// TIA Portal V19 export
DATA_BLOCK "ProcessAndPbAlarms"   // DB2
{ S7_Optimized_Access := 'TRUE' }
AUTHOR : FLA
FAMILY : UHT
VERSION : 1.0
// stored: AutoNumber false, MemoryReserve 0
   VAR
      "A" : Array[1..96] of Bool;
   END_VAR
BEGIN
   // "A"[1] : A01_TankInProcess
   // "A"[2] : A02_TankNotClean
   // "A"[3] : A03_NoInstrumentAir
   // "A"[4] : A04_NoSteam
   // "A"[5] : A05_DrainIsActive
   // "A"[6] : A06_CipFillerStarted
   // "A"[7] : A07_CipUnitOccupied
   // "A"[8] : A08_NotReadyForCip
   // "A"[9] : A09_NoProcessActive
   // "A"[10] : A10_AllreadyInStopPhase
   // "A"[11] : A11_TankIsBeingFilled
   // "A"[12] : A12_NotReadyForTotalStop
   // "A"[13] : A13_DrainTankNotAllowed
   // "A"[14] : A14_CipOnTankStared
   // "A"[15] : A15_ChainWashSelected
   // "A"[16] : A16_NoCipProgramSelected
   // "A"[17] : A17_ContinueDosingSelect
   // "A"[18] : A18_SwingbendOutOfPosn
   // "A"[19] : A19
   // "A"[20] : A20
   // "A"[21] : A21
   // "A"[22] : A22
   // "A"[23] : A23
   // "A"[24] : A24
   // "A"[25] : A25
   // "A"[26] : A26
   // "A"[27] : A27
   // "A"[28] : A28
   // "A"[29] : A29
   // "A"[30] : A30
   // "A"[31] : A31
   // "A"[32] : A32
   // "A"[33] : A33_TT0176TooLow
   // "A"[34] : A34_TT0160TooLow
   // "A"[35] : A35_TT0163TooLow
   // "A"[36] : A36_TT0178TooLow
   // "A"[37] : A37_TT0176Low
   // "A"[38] : A38_TT0178Low
   // "A"[39] : A39_TankReadyforProd
   // "A"[40] : A40_LyedosingTooLong
   // "A"[41] : A41_AcidDosingTooLong
   // "A"[42] : A42_DrainTheTank
   // "A"[43] : A43_WaitingForCipUnit
   // "A"[44] : A44_FillPressureTooLow
   // "A"[45] : A45_FillingPressureLow
   // "A"[46] : A46_LyeContainerEmpty
   // "A"[47] : A47_AcidContainerEmpty
   // "A"[48] : A48_TankEmpty
   // "A"[49] : A49_TankFull
   // "A"[50] : A50_SiemensBatteryLow
   // "A"[51] : A51_NoWater
   // "A"[52] : A52_ProdAtFillingMash
   // "A"[53] : A53_FillerNotReadyForCip
   // "A"[54] : A54_NoInstrumentAir
   // "A"[55] : A55_NoSteam
   // "A"[56] : A56
   // "A"[57] : A57_TT0951TooLow
   // "A"[58] : A58_TT0951Low
   // "A"[59] : A59_TT0950TooLow
   // "A"[60] : A60_TT0950Low
   // "A"[61] : A61_Hamba_Valve_Fault
   // "A"[62] : A62_Hamba_Barrier_low
   // "A"[63] : A63_Stop_CIP_PB_Operated
   // "A"[64] : A64_TT0178_TempFault
   // "A"[65] : A65_TT0930_Low
   // "A"[66] : A66_TT0930_Low_SIP
   // "A"[67] : A67_TT0931_Low
   // "A"[68] : A68_CT0930_High
   // "A"[69] : A69_TT0941_TempFault
   // "A"[70] : A70_TT0940_Low_Prod
   // "A"[71] : A71_TT0940_Low_SIP
   // "A"[72] : A72_TT0941_Low_SIP
   // "A"[73] : A73_CT0931_High
   // "A"[74] : A74_PG_EOL_Low_Prod
   // "A"[75] : A75_PG_EOL_Low_SIP
   // "A"[76] : A76_PG_SIP_HighTemp
   // "A"[77] : A77_PG_SIP_HighHighTemp
   // "A"[78] : A78_PG_PTX0940HighPress
   // "A"[79] : dx9_6_Spare
   // "A"[80] : dx9_7_Spare
   // "A"[81] : dx10_0_Spare
   // "A"[82] : dx10_1_Spare
   // "A"[83] : dx10_2_Spare
   // "A"[84] : dx10_3_Spare
   // "A"[85] : dx10_4_Spare
   // "A"[86] : dx10_5_Spare
   // "A"[87] : dx10_6_Spare
   // "A"[88] : dx10_7_Spare
   // "A"[89] : dx11_0_Spare
   // "A"[90] : dx11_1_Spare
   // "A"[91] : dx11_2_Spare
   // "A"[92] : dx11_3_Spare
   // "A"[93] : dx11_4_Spare
   // "A"[94] : dx11_5_Spare
   // "A"[95] : dx11_6_Spare
   // "A"[96] : dx11_7_Spare
END_DATA_BLOCK
